(* CoDeSys 2.3 library: Smi_plc.lib *)

(* Global variable list: Error_Codes *)
VAR_GLOBAL CONSTANT
	(** @name Error Return Codes SMI
		Error code MOD 1000: are the error numbers below, see Smi_ExtractLibErr()
	@{ *)
	Smi_ERC_ConnId_InUse:	DINT := 2; (**< State connection-handle in use, communication cannot be reinitialized or closed *)
	Smi_ERC_Busy:			DINT := 1; (**< State busy, wait till finished *)
	Smi_ERC_Ok:				DINT := 0; (**< State OK, block can perform new order *)
	Smi_ERC_OtherError:		DINT := -1; (**< Other error not forward *)
	Smi_ERC_ParmInvalid:	DINT := -2; (**< Parameters are invalid *)
	Smi_ERC_NoCard:			DINT := -3; (**< Card not found / existing *)
	Smi_ERC_GetModNb:		DINT := -4; (**< Can't get Module-Number *)
	Smi_ERC_GetVal:			DINT := -5; (**< GetValue unsuccessfull *)
	Smi_ERC_SetVal:			DINT := -6; (**< SetValue unsuccessfull *)
	Smi_ERC_NoHandle:		DINT := -7; (**< Invalid Connection/Handle *)
	Smi_ERC_NoSelf:			DINT := -8; (**< User not identified as PLC project *)
	Smi_ERC_NoMemory:		DINT := -10; (**< No free Memory *)
	Smi_ERC_Internal:		DINT := -11; (**< Internal error on RPC-Requester *)
	Smi_ERC_RepQAdd:		DINT := -12; (**< Reply-Queue full *)
	Smi_ERC_Timeout:		DINT := -13; (**< Communication time exceeded/Communication timeout *)
	Smi_ERC_SendCall:		DINT := -14; (**< Can't send request *)
	Smi_ERC_GetBlk:			DINT := -15; (**< GetBlock unsuccessfull *)
	Smi_ERC_SetBlk:			DINT := -16; (**< SetBlock unsuccessfull *)
	Smi_ERC_GetFnLib:		DINT := -17; (**< Can't get Function-Library *)
	Smi_ERC_WrongVers:		DINT := -18; (**< Wrong Version of MSys *)
	Smi_ERC_ResultLen:		DINT := -19; (**< Reply-Size does not match *)
	Smi_ERC_GetValLst:		DINT := -20; (**< GetValLst unsuccessfull *)
	Smi_ERC_SetValLst:		DINT := -21; (**< SetValLst unsuccessfull *)
	Smi_ERC_GetAddr:		DINT := -22; (**< GetAddress unsuccessfull *)
	Smi_ERC_ModInfo:		DINT := -24; (**< ModInfo-Rpc unsuccessfull *)
	Smi_ERC_AppInfo:		DINT := -25; (**< AppInfo-Rpc unsuccessfull *)
	Smi_ERC_SemCreate:		DINT := -26; (**< Failed to create semaphore *)
	Smi_ERC_PingInternal:	DINT := -30; (**< Intenal Error execute Ping *)
	Smi_ERC_RequestAccess:  DINT := -31; (**< RequestAccess-Rpc unsuccessfull *)
	Smi_ERC_ReleaseAccess:  DINT := -32; (**< RequestAccess-Rpc unsuccessfull *)
	Smi_ERC_LoginFail:		DINT := -95; (**< Authentification fail Name/Passwd *)
	(** @} *)

	(** @name Error Return Codes SVI
		Error code / -1000: SVI error number of counterpart, see Smi_ExtractSmiErr()
	@{ *)
	SVI_ERC_OK: 			DINT := 16#0; (**< O.K. *)
	SVI_ERC_UNDEF: 			DINT := 16#124; (**< FUNCTION NOT supported *)
	SVI_ERC_ADDR: 			DINT := 16#130; (**< SVI address NOT valid *)
	SVI_ERC_WRITE: 			DINT := 16#141; (**< SVI value NOT writable *)
	SVI_ERC_READ: 			DINT := 16#140; (**< SVI value NOT readable *)
	SVI_ERC_FAILED: 		DINT := 16#100; (**< Unspecified error *)
	SVI_ERC_OLDADDR: 		DINT := 16#17E; (**< Address NOT valid anymore *)
	SVI_ERC_NOMOD: 			DINT := 16#129; (**< Module NOT found *)
	SVI_ERC_BADNAME: 		DINT := 16#137; (**< Invalid varibale name *)
	SVI_ERC_PARM: 			DINT := 16#110; (**< Parameter NOT valid *)
	SVI_ERC_VARINUSE: 		DINT := 16#1AC; (**< Varibale already in use *)
	SVI_ERC_MBTRANS: 		DINT := 16#1AD; (**< This needs MB support *)
	SVI_ERC_MBNOBUFF: 		DINT := 16#1AE; (**< No buffer found *)
	SVI_E_NOMEM:            DINT := 16#123; (**< Not enough memory *)
	SVI_E_BADUSERLVL:  		DINT := 16#1EA; (**< Weak user level (deprecated: replaced by SVI_E_ACCDENIED) *)
	SVI_E_BADRANGE:     	DINT := 16#17C; (**< SVI value out of bounds *)
	SVI_E_ACCDENIED:    	DINT := 16#1E9; (**< Access denied *)
	SVI_E_DSIZE:        	DINT := 16#1C2; (**< Data size not valid, exceeds max size *)
	SVI_E_REDULOCK:     	DINT := 16#1F0; (**< Write access allowed only on primary CPU *)
	SVI_E_BADTYPE:      	DINT := 16#16A; (**< Wrong data type *)
	SVI_E_DLEN:         	DINT := 16#1F3; (**< Data length invalid *)
	SVI_E_BADSESS:          DINT := 16#19C; (**< Session ID not valid *)
	SBI_E_TIMEOUT2:         DINT := 16#127; (**< No answer from SW-Module *)
	(** @} *)

	(** @name Error Return Codes Socket-FBs
		Error code MOD 1000: are the error numbers below, see Smi_ExtractLibErr() \n
		Error code / -1000: VxWorks error number of the C function, see errno.h, Smi_ExtractSmiErr()
	@{ *)
	Smi_ERC_SockCreate:		DINT := -1; (**< Creation of socket failed *)
	Smi_ERC_SockClose:		DINT := -2; (**< Close of socket failed *)
	Smi_ERC_SockRead:		DINT := -3; (**< Read of socket failed *)
	Smi_ERC_SockWrite:		DINT := -4; (**< Write of socket failed *)
	Smi_ERC_SockBind:		DINT := -5; (**< bind of socket failed *)
	Smi_ERC_SockListen:		DINT := -6; (**< listen at socket init failed *)
	Smi_ERC_SockAccept:		DINT := -7; (**< accept at socket init failed *)
	Smi_ERC_SockConnect:	DINT := -8; (**< Connect failed *)
	Smi_ERC_SockInvProt:	DINT := -9; (**< Invalid protocoll *)
	Smi_ERC_SockShutdown:	DINT := -10; (**< Shutdown failed *)
	Smi_ERC_SockSetOpt:		DINT := -11; (**< Set option of socket failed *)
	(** @} *)

	(** @name Error Return Codes Retain
		for Smi_RetainExport() or its SMI-Call
	@{ *)
	RETEXP_E_UNKNOWNERROR: 		DINT := 100; (**< Unexpected error. *)
	RETEXP_E_NOMEMORY: 			DINT := 102; (**< Not enough memory. *)
	RETEXP_E_MISSINGSTRUCTFILE: DINT := 103; (**< The retain structure couldn't be found. *)
	RETEXP_E_MISSINGDATAFILE: 	DINT := 104; (**< The retain data couldn't be found. *)
	RETEXP_E_RETAINDATACORRUPT: DINT := 105; (**< The retain data is corrupt. *)
	RETEXP_E_FILECREATIONFAILED:DINT := 106; (**< The export file couldn't be created/overwritten. *)
	(** @} *)
END_VAR

(* Global variable list: Global_Constants *)
(*
 PLC1131-Library with Functions for Communication by SVI and SMI
 Copyright: G.Bachmann GmbH, 1997-2011, Feldkirch - Austria
*)
VAR_GLOBAL CONSTANT
	(** @name Constants for 'VarCode'
	@{ *)
	Smi_MX_Code:			INT := 1; (**< MX marker *)
	Smi_MB_Code:			INT := 2; (**< MB marker *)
	Smi_MD_Code:			INT := 3; (**< MD marker *)
	Smi_MR_Code:			INT := 4; (**< MR marker *)
	Smi_MW_Code:			INT := 5; (**< MW marker *)
	Smi_RD_Code:			INT := 19; (**< RD marker *)
	Smi_GD_Code:			INT := 35; (**< GD marker *)
	(** @} *)

	(** @name Constants for 'ProtVers'
		in SMI_Connect(), SMI_Connect_NB(), SMI_Login(), SMI_Login_NB() and SMI_Ping() 
	@{ *)
	Smi_PROT_Tcp:			DWORD := 16#80000000; (**< Use TCP instead of UDP *)
	Smi_PROT_QSoap:			DWORD := 16#00004000; (**< Use bachmann proprietary SOAP as transport protocol (Quick SOAP)*)
	Smi_PROT_Ssl:           DWORD := 16#08000000; (**< Use SSL transport protocol *)
	Smi_PROT_PlainTxtPwd:   DWORD := 16#04000000; (**< Send plain text password *)
	(** @} *)

	(** @name Constants for 'TestLevel' and 'TestResult'
		in SMI_Ping(), SMI_PingEx()
	@{ *)
	Smi_LEVEL_IpPing:		WORD := 1; (**< IP-Ping *)
	Smi_LEVEL_AppInfo:		WORD := 2; (**< RES_APPINFO-Rpc *)
	Smi_LEVEL_ModInfo:		WORD := 4; (**< RES_MODINFO-Rpc *)
	Smi_LEVEL_RpcPing:		WORD := 8; (**< Rpc-Ping to Module *)
	Smi_LEVEL_FtpCheck:		WORD := 16; (**< Ftp-Test-Login *)
	(** @} *)

	(** @name Constants for 'AppState'
		in SMI_Ping(), SMI_PingEx()
	@{ *)
	Smi_RESSTAT_Run:		DWORD := 1; (**< Module is running *)
	Smi_RESSTAT_Error:		DWORD := 2; (**< Module is in error *)
	Smi_RESSTAT_Stop:		DWORD := 3; (**< Module stopped *)
	Smi_RESSTAT_Init:		DWORD := 4; (**< Module is in init *)
	Smi_RESSTAT_Deinit:		DWORD := 5; (**< Module is in deinit *)
	Smi_RESSTAT_Eoi:		DWORD := 6; (**< Module is waiting *)
	(** @} *)

	(** @name Available SMI Commands
		of SMI_Command()
	@{ *)
	CMD_SMI_PROC_NULL:			DWORD := 0; (**< SMI-Ping *)
	CMD_SMI_PROC_DEINIT:		DWORD := 4; (**< Uninstall module *)
	CMD_SMI_PROC_RESET:			DWORD := 6; (**< Reset module *)
	CMD_SMI_PROC_NEWCFG:		DWORD := 8; (**< New configuration of module *)
	CMD_SMI_PROC_ENDOFINIT:		DWORD := 14; (**< Signal end of init *)
	CMD_SMI_PROC_STOP:			DWORD := 18; (**< Stop module *)
	CMD_SMI_PROC_RUN:			DWORD := 20; (**< Start module *)
    CMD_PLC_PROC_RETAINEXPORT:  DWORD := 1546; (**< Export RETAIN data FOR an application *)
	(** @} *)

	(** @name Constants of Sockets
		of Smi_SOCK_ClientOpen(), Smi_SOCK_ClientOpen_NB(), Smi_SOCK_ServerOpen(), Smi_SOCK_ServerOpen_NB()
	@{ *)
	Smi_SOCK_ProtoTCP:		DWORD :=  6; (**< Protocol AF_INET/TCP *)
	Smi_SOCK_ProtoUDP:		DWORD := 17; (**< Protocol AF_INET/UDP *)
	Smi_SOCK_ModeDirect:	DINT := 0; (**< Parameter for mode: direct operation *)
	Smi_SOCK_ModeNoWait:	DINT := 2; (**< Parameter for mode: Smi_SOCK_Read() returns immediatly *)
	Smi_SOCK_SO_KEEPALIVE:	DINT := 16#0008; (**< keep connections alive, 1(on=default)/0(off) *)
 	Smi_SOCK_SO_BROADCAST:	DINT := 16#0020; (**< permit sending to multiple destination 1(on)/0(off) *)
 	Smi_SOCK_SO_SNDBUFF:	DINT :=	16#1001; (**< specifying the size of the send buffer *)
 	Smi_SOCK_SO_RCVBUFF:	DINT := 16#1002; (**< specifying the size of the beceive buffer *)
	(** @} *)
END_VAR

(* Global variable list: Library_Info *)
VAR_GLOBAL CONSTANT
	SMI_PLC_LIBVER					:	STRING(16) 	:=	'V1.36 Release';	(* Version String *)
    SMI_PLC_MMPREADY                :   BOOL        :=  TRUE;               (* MMP Ready *)
END_VAR

(* Data type *)
(*
	structure to specify 64 Bit Smi Address Handle
*)
TYPE SMI_ADDR
STRUCT
	Addr1:		DWORD;		(* SmiAddr Handle 1st 32 Bit *)
	Addr2:		DWORD;		(* SmiAddr Handle 2nd 32 Bit *)
END_STRUCT
END_TYPE

(* Data type *)
(*
	return-structure of Smi_GetConnStatus
*)
TYPE SMI_RETCONNSTAT
STRUCT
	RetCode:	DINT;		(* Success (0) - or Error-Code (<0) *)
	CpuNb:		DINT;		(* CPU-Number *)
	ModuleNb:	DWORD;		(* Module-Number (SMI-Master) *)
	PLibAddr:	DWORD;		(* SVI-Function-Lib-Pointer *)
	UseCount:	DINT;		(* Number of pending requests (FBs) *)
	ErrorCode:	DINT;		(* Last Error on Connection *)
	FnGetStat:	DINT;		(* Read/Write-Get-Status *)
	FnRdyStat:	DINT;		(* Read/Write-Ready-Status *)
END_STRUCT
END_TYPE

(* Data type *)
(* This structure is filled at Smi_SOCK_ClientOpen and
   Smi_SOCK_ServerOpen *)
TYPE SMI_SOCK_CONTROL :
STRUCT
	ProtType:		DWORD;
	Port:			WORD;
	IpAddr:			DINT;
	Socket:			DWORD;
    ServerSocket:   DWORD;
END_STRUCT
END_TYPE

(* Data type *)
(*
	structure to specify a Marker-Variable
*)
TYPE VAR_ADDR
STRUCT
	VarCode:	DWORD;		(* Marker-Type 1:MX, 2:MB, 3:MD, 4:MR, 5:MW *)
	VarIndex:	DWORD;		(* Index of Marker *)
END_STRUCT
END_TYPE

(* POU GetREALasDWORD, IL *)
(**
@brief Return a REAL from contents of DWORD
@param[in] dw Input variable
@return REAL interpreted value
*)
FUNCTION GetREALasDWORD : REAL
VAR_INPUT
	dw: DWORD;
END_VAR
	LD		0
END_FUNCTION

(* POU SetREALasDWORD, IL *)
(**
@brief Returns REAL 'x' casted to a DWORD
@param[in] x REAL value
@return DWORD-coded value
*)
FUNCTION SetREALasDWORD : DWORD
VAR_INPUT
	x: REAL;
END_VAR
LD 0
END_FUNCTION

(* POU Smi_BuildNbFromIP, IL *)
(**
@brief Makes a CPU-Number representing an IP-Address
@param[in] b1 1. Byte of the IP adress
@param[in] b2 2. Byte of the IP adress
@param[in] b3 3. Byte of the IP adress
@param[in] b4 4. Byte of the IP adress
@return Coded IP address (CPU number)
*)
FUNCTION Smi_BuildNbFromIP : DINT
VAR_INPUT
	b1: BYTE;
	b2: BYTE;
	b3: BYTE;
	b4: BYTE;
END_VAR
LD 0
END_FUNCTION

(* POU Smi_BuildNbFromName, IL *)
(**
@brief Makes a CPU-Number for a Host-Name or an IP-String
@param[in] Name IP-Adresse in octet-Notation (e.g. 192.9.200.30)
@return Coded IP address (CPU number). The value is to be transferred 
	to the input parameter CpuNb of the function blocks SMI_Connect() and SMI_CheckIp_NB appropriate. 
*)
FUNCTION Smi_BuildNbFromName : DINT
VAR_INPUT
	Name : STRING(23);
END_VAR
	LD		0
END_FUNCTION

(* POU SMI_BuildNbFromName_NB, ST *)
(**
@brief Makes a CPU-Number for a Host-Name or an IP-String, non-blocking.
@param[in] Req If false only state is returned. If true and state is not busy,
    a command is done.
@param[in] Name IP-Address in Octet-Notation  '192.9.100.10' or 'hostname'
@param[out] Done TRUE if ready
@param[out] Error TRUE in case of error
@param[out] Status Error code in case of error 
    - <tt>#Smi_ERC_Ok</tt>OK. <tt>Done = TRUE</tt>, <tt>ConnId</tt> valid
    - <tt>#Smi_ERC_Busy</tt>Completion/response is pending, <tt>CpuNb </tt> is not available
    - <tt>#Smi_ERC_OtherError</tt>Name or IP address is invalid, CpuNb is not available.
@param[out] CpuNb Coded IP address (CPU number). The value is to be transferred to the input 
	parameter CpuNb of the function blocks SMI_Connect(), SMI_Connect_NB(), SMI_Login(), SMI_Login_NB() 
	and SMI_CheckIp_NB appropriate.
*)
FUNCTION_BLOCK SMI_BuildNbFromName_NB
VAR_INPUT
	Req:			BOOL;
    Name:       	STRING(63);
END_VAR
VAR_OUTPUT
	Done: 		BOOL;
	Error: 		BOOL;
	Status: 	DINT;
	CpuNb: 		DINT;
END_VAR
VAR
	Pltd: DWORD;
END_VAR
;
END_FUNCTION_BLOCK

(* POU SMI_Call, IL *)
(**
@brief This function block is used to send SMI-messages. Timeout is
    interal set to 2000ms and no retries.
  Note: The size of the in and out buffer are limited to SMI_DATALEN.
@param[in] Req If false only state is returned. If true and state is not busy,
    a command is done.
@param[in] ConnId Connection identifier for the connection. 
           The connection identifier can be determined with SMI_Login() or SMI_Connect().
@param[in] SmiFcnNumber Specifies which SMI functions should be executed. 
    General SMI functions can be called
@param[in] DataSend Address of send buffer, use ADR(). Specification of the transmit 
    buffer Maximum size: 1996 bytes.
@param[in] DataSendLen Length of send buffer. 
    Specification of the transmit buffer Maximum size: 1996 bytes. 
@param[in] DataRec Address of receive buffer, use ADR(). 
    Specification of the receive buffer Maximum size: 1996 bytes. 
@param[in] DataRecLen Specification of the receive buffer Maximum size: 1996 bytes.
@param[out] State Error code in case of error 
    - <tt>#Smi_ERC_Ok</tt> OK
    - <tt>#Smi_ERC_Busy</tt> Completion/response is pending
    - <tt>Smi_ERC_*</tt> Error codes are negative
@param[out] RecLen Specification of the number of bytes received
    The minimum of <tt>DataRecLen</tt> and RecLen is copied to the receive buffer.
*)
FUNCTION_BLOCK SMI_Call
VAR_INPUT
	Req:			BOOL;
	ConnId:			DWORD;
	SmiFcnNumber:	DWORD;
	DataSend:		DWORD;
	DataSendLen:	DINT;
	DataRec:		DWORD;
	DataRecLen:		DINT;
END_VAR
VAR_OUTPUT
	State: 			DINT;
	RecLen:			DINT;
END_VAR
VAR
	fi: 			UDINT;
END_VAR
	LD		0
END_FUNCTION_BLOCK

(* POU SMI_CheckIp_NB, ST *)
(**
@brief non-blocking FB to check if an IP is occupied. (on MPC only)
@param[in] Req Request enable
@param[in] EthCard To use Ethernet interface (starting with 0).
@param[in] CpuNb Coded IP address (CPU number).\n
    The IP address must be coded beforehand. (Smi_BuildNbFromIP or Smi_BuildNbFromName). 
@param[in] Timeout The parameter is used to indicate the response latency. By Timeout = 0 
	is wait for 3 seconds. [ms]
@param[out] Mac Contains the MAC address of the desired host when parameter Done is set.
@param[out] MacHexStr Contains the MAC address in string format when parameter Done is set.
@param[out] Done TRUE if ready
@param[out] Error TRUE in case of error
@param[out] Status Error code in case of error 
    - <tt>#Smi_ERC_Ok</tt> OK. <tt>Done = TRUE</tt>, <tt>Mac</tt> valid
    - <tt>#Smi_ERC_Busy</tt> Completion/response is pending, <tt>Mac</tt> is not available
    - <tt>Smi_ERC_*</tt> Error codes are negative. <tt>Error = TRUE;</tt> Mac not available. 
*)
FUNCTION_BLOCK SMI_CheckIp_NB
VAR_INPUT
	Req: BOOL;
	EthCard: DINT;
	CpuNb: DINT;
	Timeout: TIME;
END_VAR
VAR_OUTPUT
	Mac: ARRAY[1..6] OF BYTE;
	MacHexStr: STRING(17);
	Done: BOOL;
	Error: BOOL;
	Status: DINT;
END_VAR
VAR
	hJob: DWORD;
END_VAR
;
END_FUNCTION_BLOCK

(* POU SMI_CloseConnect, ST *)
(**
@brief close a connection to a remote host opened with SMI_Connect or SMI_Login
@param[in] Req Request enable
@param[in] ConnId Transfer of the connection identifier for the connection.
    The identifier can be determined with SMI_Login() or SMI_Connect().
@param[out] Done TRUE if ready
@param[out] Error TRUE in case of error
@param[out] Status Error code in case of error
    - <tt>#Smi_ERC_Ok</tt> OK. <tt>Done = TRUE</tt>
    - <tt>Smi_ERC_*</tt> Error codes are negative
*)
FUNCTION_BLOCK SMI_CloseConnect
VAR_INPUT
	Req: BOOL;
	ConnId: DWORD;
END_VAR
VAR_OUTPUT
	Done: BOOL;
	Error: BOOL;
	Status: DINT;
END_VAR
VAR
END_VAR
;
END_FUNCTION_BLOCK

(* POU SMI_Command, IL *)
(**
@brief This function block is used to send SMI-messages. Timeout is
    interal set to 2000ms and no retries.
@param[in] Req request-enable: if false only state is returned
@param[in] ConnId Connection identifier for the connection. 
           The connection identifier can be determined with SMI_Login() or SMI_Connect().
@param[in] SmiFcnNumber SMI function to be executed. Allowed functions
    - <tt>#CMD_SMI_PROC_NULL</tt>
    - <tt>#CMD_SMI_PROC_DEINIT</tt>
    - <tt>#CMD_SMI_PROC_RESET</tt>
    - <tt>#CMD_SMI_PROC_NEWCFG</tt>
    - <tt>#CMD_SMI_PROC_ENDOFINIT</tt>
    - <tt>#CMD_SMI_PROC_STOP</tt>
    - <tt>#CMD_SMI_PROC_RUN</tt>
@param[in] ModuleName Name of target module, has to be the same as in SMI_Connect or
    SMI_Login
@param[out] Error If TRUE error occured
@param[out] State Error code in case of error 
    - <tt>#Smi_ERC_Ok</tt> OK
    - <tt>#Smi_ERC_Busy</tt> Completion/response is pending
    - <tt>Smi_ERC_*</tt> Error codes are negative
*)
FUNCTION_BLOCK SMI_Command
VAR_INPUT
	Req			: BOOL;
	ConnId		: DWORD;
	SmiFcnNumber :	DWORD;
	ModuleName 	: STRING(11);
END_VAR
VAR_OUTPUT
	Error	 	: BOOL;
	State	 	: DINT;
END_VAR
VAR
	fi: UDINT;
END_VAR
	LD		0
END_FUNCTION_BLOCK

(* POU SMI_Connect, IL *)
(**
@brief Build/init Connection to named SMI-Module on local or remote CPU
@param[in] CpuNb With the parameter the IP address of the CPU of the communication partner will be transferred. 
@param[in] MasterName With the parameter, the name of the partner module (communication partner) will be transferred.
@param[in] Reinit The parameter must be set if a previously-established connection should be renewed
@param[in] ProtVers The parameter is used to specify the RPC protocol version to be used. This input must be used 
	when SMI is used for the connection.
    The possible RPC protocol versions depend on the communication partner (process value supplier). This input can 
	be used to switch the protocol to TCP using the entry SMI_PROT_Tcp (OR link with the protocol version). The UDP 
	protocol is used without OR link with PROT_Tcp. System modules/handler and PLC projects based on M1 software 
	V1.00 release and the simultaneously-created available controller modules generally use RPC protocol version 2. 
	Consequently, the value 2 has to be indicated at the parameter ProtVers.
@param[out] Done TRUE if ready
@param[out] Error TRUE in case of error
@param[out] Status Error code in case of error
    - <tt>#Smi_ERC_Ok</tt> OK. <tt>Done = TRUE</tt>, <tt>ConnId</tt> valid
    - <tt>#Smi_ERC_Busy</tt> Completion/response is pending, <tt>ConnId</tt> is not available
    - <tt>#Smi_ERC_ConnId_InUse</tt> Reinitialization presently not possible; communication in process
    - <tt>Smi_ERC_*</tt> Error codes are negative. 
@param[out] ConnId Connection-Identifier
*)
FUNCTION_BLOCK SMI_Connect
VAR_INPUT
	CpuNb: 		DINT;
	MasterName: STRING(15);
	Reinit: 	BOOL;
	ProtVers: 	DWORD;
END_VAR
VAR_OUTPUT
	Done: 		BOOL;
	Error: 		BOOL;
	Status: 	DINT;
	ConnId: 	DWORD;
END_VAR
VAR
	fi: UDINT;
END_VAR
LD 0
END_FUNCTION_BLOCK

(* POU SMI_Connect_NB, IL *)
(**
@brief Non blocking version of SMI_Connect, Build/init Connection to named SMI-Module on local or remote CPU
@param[in] CpuNb With the parameter the IP address of the CPU of the communication partner will be transferred.
    see Smi_BuildNbFromName()
@param[in] MasterName With the parameter, the name of the partner module (communication partner) will be transferred.
@param[in] Reinit The parameter must be set if a previously-established connection should be renewed
@param[in] ProtVers The parameter is used to specify the RPC protocol version to be used. This input 
	must be used when SMI is used for the connection.\n
    The possible RPC protocol versions depend on the communication partner (process value supplier). This input can 
	be used to switch the protocol to TCP using the entry SMI_PROT_Tcp (OR link with the protocol version). The UDP 
	protocol is used without OR link with PROT_Tcp. System modules/handler and PLC projects based on M1 software 
	V1.00 release and the simultaneously-created available controller modules generally use RPC protocol version 2. 
	Consequently, the value 2 has to be indicated at the parameter ProtVers.
@param[out] Done TRUE if ready
@param[out] Error TRUE in case of error
@param[out] Status Error code in case of error
    - <tt>#Smi_ERC_Ok</tt> OK. <tt>Done = TRUE</tt>, <tt>ConnId</tt> valid
    - <tt>#Smi_ERC_Busy</tt> Completion/response is pending, <tt>ConnId</tt> is not available
    - <tt>#Smi_ERC_ConnId_InUse</tt> Reinitialization presently not possible; communication in process
    - <tt>Smi_ERC_*</tt> Error codes are negative. 
@param[out] ConnId Connection-Identifier
*)
FUNCTION_BLOCK SMI_Connect_NB
VAR_INPUT
	CpuNb: 		DINT;
	MasterName: STRING(15);
	Reinit: 	BOOL;
	ProtVers: 	DWORD;
END_VAR
VAR_OUTPUT
	Done: 		BOOL;
	Error: 		BOOL;
	Status: 	DINT;
	ConnId: 	DWORD;
END_VAR
VAR
	fi: UDINT;
	Pltd: DWORD;
	uState: DWORD;
END_VAR
LD 0
END_FUNCTION_BLOCK

(* POU Smi_ExtractLibErr, ST *)
(**
@brief The functions and functionblocks of the SMI-library return
    a 'packed' error-code/status which encodes two specific errors.

    This function extracts the library-error of the encoded error.
    The library-error is generated in the SMI-library directly,
    eg through checking the input-parameters.

    The library-error can be compared against the Smi_ERC_xxx-constants.

@param[in] Error Error returned by the Smi_-function or -functionblock
@return DINT, see description
*)
FUNCTION Smi_ExtractLibErr : DINT
VAR_INPUT
	Error: DINT;
END_VAR
VAR
END_VAR
;
END_FUNCTION

(* POU Smi_ExtractSmiErr, ST *)
(**
@brief Functions and functions of the SMI-library, return
    a 'packed' error-code/status which encodes two specific errors.

    This function extracts the SMI-error (error/return-value
    of the SMI-reply-message) of the encoded error.
@param[in] Error error returned by the Smi_-function or -functionblock
@return DINT, see description
*)
FUNCTION Smi_ExtractSmiErr : DINT
VAR_INPUT
	Error: DINT;
END_VAR
VAR
END_VAR
;
END_FUNCTION

(* POU SMI_GetAddr, ST *)
(**
@brief Gets the SMI-Address-Handle of the Symbolic SVI-Object from
    SMI-Module
@param[in] Req Request enable
@param[in] ConnId Transfer of the connection identifier for the connection. 
    The identifier can be determined with SMI_Login() or SMI_Connect(). 
@param[in] ValueName With the parameter the symbolic marker or process value 
    name is specified, for which the numeric address should be determined.
@param[out] Ndr TRUE if operation successfully completed/new data received
@param[out] Error TRUE in case of error
@param[out] Status see Smi_ERC_*
    - #Smi_ERC_Ok OK/Done
    - #Smi_ERC_Busy Completion/response is pending, result is not available
    - Smi_ERC_* Error occured
@param[out] Error TRUE in case of error
@param[out] SmiHandle Smi-Address-Handle of the Symbolic Object
*)
FUNCTION_BLOCK SMI_GetAddr
VAR_INPUT
	Req 		: BOOL;
	ConnId 		: DWORD;
	ValueName 	: STRING(63);
END_VAR
VAR_OUTPUT
	Ndr 		: BOOL;
	Error 		: BOOL;
	Status 		: DINT;
	SmiHandle	: SMI_ADDR;
END_VAR
VAR
	fi			: UDINT;
END_VAR
;
END_FUNCTION_BLOCK

(* POU SMI_GetAddress, ST *)
(**
@brief Gets Address of a Marker or Process-Value from SMI-Module
@param[in] Req Request enable
@param[in] ConnId Transfer of the connection identifier for the connection.
    The identifier can be determined with SMI_Login() or SMI_Connect().
@param[in] ValueName With the parameter the symbolic marker or process value name is specified, for which 
	the numeric address should be determined.
@param[out] Ndr TRUE if new data received
@param[out] Error TRUE in case of error
@param[out] Status Error code in case of error
    - <tt>#Smi_ERC_Ok</tt> OK. <tt>Ndr = TRUE</tt>, <tt>VAddr</tt> valid
    - <tt>#Smi_ERC_Busy</tt> Completion/response is pending, <tt>VAddr</tt> is not available
    - <tt>#Smi_ERC_ConnId_InUse</tt> Reinitialization presently not possible; communication in process
    - <tt>Smi_ERC_*</tt> Error codes are negative
@param[out] VAddr Marker- or Process-Value-Address
*)
FUNCTION_BLOCK SMI_GetAddress
VAR_INPUT
	Req : BOOL;
	ConnId : DWORD;
	ValueName : STRING(63);
END_VAR
VAR_OUTPUT
	Ndr : BOOL;
	Error : BOOL;
	Status : DINT;
	VAddr : VAR_ADDR;
END_VAR
VAR
	fi: UDINT;
END_VAR
;
END_FUNCTION_BLOCK

(* POU SMI_GetBlk, ST *)
(**
@brief Reads a String or Stream of Bytes from SMI-Module
@param[in] Req Request enable
@param[in] ConnId Transfer of the connection identifier for the connection.
    The identifier to be transferred can be determined with SMI_Login() or SMI_Connect().
@param[in] SmiHandle The start address of the marker block to be read or the SVI variable.
    This is determined by SMI_GetAddr().
@param[in] Addr Address of a data range into which the values are read.
@param[in] Length Length of the data range. If a block of markers is read, the value byte 
	stream is 4 byte aligned. 
@param[out] Ndr TRUE if operation successfully completed/new data received
@param[out] Error TRUE in case of error
@param[out] Status see Smi_ERC_*
    - #Smi_ERC_Ok OK/Done
    - #Smi_ERC_Busy Completion/response is pending, result is not available
    - Smi_ERC_* Error occured
@param[out] NRead number of bytes read
*)
FUNCTION_BLOCK SMI_GetBlk
VAR_INPUT
	Req			: BOOL;
	ConnId		: DWORD;
	SmiHandle	: SMI_ADDR;
	Addr 		: DWORD;
	Length		: UINT;
END_VAR
VAR_OUTPUT
	Ndr			: BOOL;
	Error	 	: BOOL;
	Status		: DINT;
	NRead		: UINT;
END_VAR
VAR
	fi			: UDINT;
END_VAR
;
END_FUNCTION_BLOCK

(* POU Smi_GetConnStatus, IL *)
(**
@brief Gets information on Status of Connection
@param[in] ConnId Transfer of the connection identifier for the connection. The identifier can be determined 
	with SMI_Login() or SMI_Connect(). 
@retval SMI_RETCONNSTAT.RetCode = #Smi_ERC_Ok: Everything OK.
@retval SMI_RETCONNSTAT.RetCode = #Smi_ERC_NoSelf: User not identified as PLC project.
*)
FUNCTION Smi_GetConnStatus : SMI_RETCONNSTAT
VAR_INPUT
	ConnId: DWORD;
END_VAR
LD 0
END_FUNCTION

(* POU Smi_GetOwnIPAddr, IL *)
(**
@brief Makes a Number representing the own IP-Address
@param[in] EthCard ethernet-interface (0 or 1)
@return Coded IP address (CPU number)
*)
FUNCTION Smi_GetOwnIPAddr : DINT
VAR_INPUT
	EthCard:	DINT;
END_VAR
LD 0
END_FUNCTION

(* POU SMI_GetVal, ST *)
(**
@brief Reads a single SVI-Var-Object from a SMI-Module
@param[in] Req Request enable
@param[in] ConnId Transfer of the connection identifier for the connection.
    The identifier to be transferred can be determined with SMI_Login() or SMI_Connect().
@param[in] SmiHandle 64-Bit Smi Object Handle/process value's address
    This is determined by SMI_GetAddr().
@param[out] Ndr TRUE if operation successfully completed/new data received
@param[out] Error TRUE in case of error
@param[out] Status see Smi_ERC_*
    - #Smi_ERC_Ok OK/Done
    - #Smi_ERC_Busy Completion/response is pending, result is not available
    - Smi_ERC_* Error occured
@param[out] Value Read-Value 32-Bit Format
*)
FUNCTION_BLOCK SMI_GetVal
VAR_INPUT
	Req			: BOOL;
	ConnId		: DWORD;
	SmiHandle	: SMI_ADDR;
END_VAR
VAR_OUTPUT
	Ndr			: BOOL;
	Error		: BOOL;
	Status		: DINT;
	Value		: DWORD;
END_VAR
VAR
	fi			: UDINT;
END_VAR
;
END_FUNCTION_BLOCK

(* POU Smi_GetValFn, IL *)
(**
@brief Reads Smi Objekt (specified by Smi Address) from SMI-Module.
    Implementation: an Rpc-Request is done, read may be BUSY
    until Rpc-Reply is received.
@param[in] ConnId Transfer of the connection identifier for the connection.
    The identifier to be transferred can be determined with SMI_Login() or SMI_Connect().
@param[in] SmiAddr Address of 64-Bit Smi Object Handle/process value's address
@param[in] ValAddr Address to store read Value
@retval #Smi_ERC_Ok OK
@retval #Smi_ERC_Busy Completion/response is pending; read value not available yet
@retval #Smi_ERC_ConnId_InUse Other function is being processed; communication in process
@retval Smi_ERC_* Error codes are negative 
*)
FUNCTION Smi_GetValFn : DINT
VAR_INPUT
	ConnId		: DWORD;
	SmiAddr		: DWORD;
	ValAddr		: DWORD;
END_VAR
LD 0
END_FUNCTION

(* POU SMI_GetValLst, IL *)
(**
@brief Reads a List of Smi-Objects from SMI-Module
@param[in] Req Request enable
@param[in] ConnId Transfer of the connection identifier for the connection.
    The identifier to be transferred can be determined with SMI_Login() or SMI_Connect().
@param[in] SmiHandleF List of Smi-Address-Handles. This is determined by SMI_GetAddr(). 
@param[in] NumberOf Number of addresses, maximal 64
@param[out] Ndr TRUE if operation successfully completed/new data received
@param[out] Error TRUE in case of error
@param[out] Status see Smi_ERC_*
    - #Smi_ERC_Ok OK/Done
    - #Smi_ERC_Busy Completion/response is pending, result is not available
    - Smi_ERC_* Error occured
@param[out] Rdf Data receive field
*)
FUNCTION_BLOCK SMI_GetValLst
VAR_INPUT
	Req			: BOOL;
	ConnId		: DWORD;
	SmiHandleF  : ARRAY[0..63] OF SMI_ADDR;
	NumberOf 	: DINT;
END_VAR
VAR_OUTPUT
	Ndr			: BOOL;
	Error	 	: BOOL;
	Status	 	: DINT;
	Rdf 		: ARRAY[0..63] OF DWORD;
END_VAR
VAR
	fi: UDINT;
END_VAR
LD 0
END_FUNCTION_BLOCK

(* POU Smi_GetVersion, ST *)
(**
@brief Returns the version string of the library. In simulation always
    '' is returned.
@param[in] dummy Unused parameter. 
@return Version string of the PLC library, e.g. V 1.03.01 Alpha, V 1.06.04 Beta, V1.04 Release.
*)
FUNCTION Smi_GetVersion : STRING(15)
VAR_INPUT
	dummy:		BOOL;
END_VAR
VAR
END_VAR
Smi_GetVersion := '';
END_FUNCTION

(* POU SMI_Login, IL *)
(**
@brief Build/init Connection to named SMI-Module with login on local 
    or remote CPU.
@param[in] CpuNb With the parameter the IP address of the CPU of the communication partner will be transferred. \n
    see: Smi_BuildNbFromName()
@param[in] MasterName With the parameter, the name of the partner module (communication partner) will be transferred.
@param[in] Reinit The parameter must be set if a previously-established connection should be renewed
@param[in] ProtVers The parameter is used to specify the RPC protocol version to be used. 
    This input must be used when SMI is used for the connection.\n
    The possible RPC protocol versions depend on the communication partner (process value supplier). This input can 
	be used to switch the protocol to TCP using the entry SMI_PROT_Tcp (OR link with the protocol version). The UDP 
	protocol is used without OR link with PROT_Tcp. System modules/handler and PLC projects based on M1 software 
	V1.00 release and the simultaneously-created available controller modules generally use RPC protocol version 2. 
	Consequently, the value 2 has to be indicated at the parameter ProtVers.
@param[in] LoginName With the parameter the login name is transferred.
@param[in] Password With the parameter the password that belongs to the login name is transferred.
    In case of an unencrypted password (Smi_PROT_PlainTxtPwd) the maximal password len is 16 (counterpart is older 
    than MSys 3.70 R) or 32 (counterpart is above MSys 3.70 R). In Case of an encrypted password the maximal len is 39. 
@param[out] Done TRUE if ready
@param[out] Error TRUE in case of error
@param[out] Status Error code in case of error
    - <tt>#Smi_ERC_Ok</tt> OK. <tt>Done = TRUE</tt>, <tt>ConnId</tt> valid
    - <tt>#Smi_ERC_Busy</tt> Completion/response is pending, <tt>ConnId</tt> is not available
    - <tt>#Smi_ERC_ConnId_InUse</tt> Reinitialization presently not possible; communication in process
    - <tt>Smi_ERC_*</tt> Error codes are negative. 
@param[out] ConnId Connection-Identifier
*)
FUNCTION_BLOCK SMI_Login
VAR_INPUT
	CpuNb: 		DINT;
	MasterName: STRING(15);
	Reinit: 	BOOL;
	ProtVers: 	DWORD;
	LoginName:	STRING(19);
	Password:	STRING(39);
END_VAR
VAR_OUTPUT
	Done: 		BOOL;
	Error: 		BOOL;
	Status: 	DINT;
	ConnId: 	DWORD;
END_VAR
VAR
	fi: UDINT;
END_VAR
	LD		0
END_FUNCTION_BLOCK

(* POU SMI_Login_NB, IL *)
(**
@brief Non-blocking version of SMI_Login. 
    Build/init Connection to named SMI-Module with login on local or remote CPU.
@param[in] CpuNb With the parameter the IP address of the CPU of the communication partner will be transferred. \n
    see: Smi_BuildNbFromName()
@param[in] MasterName With the parameter, the name of the partner module (communication partner) will be transferred.
@param[in] Reinit The parameter must be set if a previously-established connection should be renewed
@param[in] ProtVers The parameter is used to specify the RPC protocol version to be used. 
    This input must be used when SMI is used for the connection.\n
    The possible RPC protocol versions depend on the communication partner (process value supplier). This input can 
	be used to switch the protocol to TCP using the entry SMI_PROT_Tcp (OR link with the protocol version). The UDP 
	protocol is used without OR link with PROT_Tcp. System modules/handler and PLC projects based on M1 software V1.00 
	release and the simultaneously-created available controller modules generally use RPC protocol version 2. Consequently, 
	the value 2 has to be indicated at the parameter ProtVers.
@param[in] LoginName With the parameter the login name is transferred.
@param[in] Password With the parameter the password that belongs to the login name is transferred.
    In case of an unencrypted password (Smi_PROT_PlainTxtPwd) the maximal password len is 16 (counterpart is older 
    than MSys 3.70 R) or 32 (counterpart is above MSys 3.70 R). In Case of an encrypted password the maximal len is 39. 
@param[out] Done TRUE if ready
@param[out] Error TRUE in case of error
@param[out] Status Error code in case of error
    - <tt>#Smi_ERC_Ok</tt> OK. <tt>Done = TRUE</tt>, <tt>ConnId</tt> valid
    - <tt>#Smi_ERC_Busy</tt> Completion/response is pending, <tt>ConnId</tt> is not available
    - <tt>#Smi_ERC_ConnId_InUse</tt> Reinitialization presently not possible; communication in process
    - <tt>Smi_ERC_*</tt> Error codes are negative. 
@param[out] ConnId Connection-Identifier
*)
FUNCTION_BLOCK SMI_Login_NB
VAR_INPUT
	CpuNb: 		DINT;
	MasterName: STRING(15);
	Reinit: 	BOOL;
	ProtVers: 	DWORD;
	LoginName:	STRING(19);
	Password:	STRING(39);
END_VAR
VAR_OUTPUT
	Done: 		BOOL;
	Error: 		BOOL;
	Status: 	DINT;
	ConnId: 	DWORD;
END_VAR
VAR
	fi: UDINT;
	Pltd : DWORD;
	uState: DWORD;
END_VAR
	LD		0
END_FUNCTION_BLOCK

(* POU SMI_Ping, IL *)
(**
@brief Test Communication to CPU/Host or named SMI-Module on local
    or remote CPU.
@param[in] Req Request enable
@param[in] CpuNb With the parameter the IP address of the CPU of the communication partner will be transferred.\n
    see Smi_BuildNbFromName()
@param[in] ModuleName With the parameter the IP address of the CPU of the communication partner is transferred. 
    Relevance depends on <tt>TestLevel</tt>.
@param[in] ProtVers The parameter <tt>ProtVers</tt> is used to specify the RPC protocol version used (usually 2).
@param[in] TestLevel Use this parameter to specify what should be tested, or the scope in which the test should be executed. 
    For this the constants Smi_LEVEL_* are available. These can also be combined.
@param[out] Done TRUE if ready
@param[out] Error TRUE in case of error
@param[out] Status Error code in case of error 
    - <tt>#Smi_ERC_Ok</tt> OK. <tt>Done = TRUE</tt>, Result valid
    - <tt>#Smi_ERC_Busy</tt> Completion/response is pending, Result is not available
    - <tt>#Smi_ERC_GetModNb</tt> The RES_MODNB-Rpc was not successful.
    - <tt>#Smi_ERC_Timeout</tt> The communication partner (the CPU, the HOST, the software module) does not respond or 
        cannot be accessed.
    - <tt>#Smi_ERC_WrongVers</tt> SMI_Ping() does not function with this version of MSys; SMI_Ping() cannot be used until 
        MSys = V1.02 is used.
    - <tt>#Smi_ERC_ResultLen</tt> The returned data is inadequate or incompletely received.
    - <tt>#Smi_ERC_ModInfo</tt> The RES_MODINFO-Rpc was not successful.
    - <tt>#Smi_ERC_AppInfo</tt> The RES_APPINFO-Rpc was not successful.
@param[out] TestResult Degree of successfull Test: <tt>Smi_LEVEL_*</tt>
@param[out] AppState State of Module or Application <tt>Smi_RESSTAT_*</tt>
*)
FUNCTION_BLOCK SMI_Ping
VAR_INPUT
	Req: BOOL;
	CpuNb: DINT;
	ModuleName: STRING(15);
	ProtVers: DWORD;
	TestLevel: WORD;
END_VAR
VAR_OUTPUT
	Done: BOOL;
	Error: BOOL;
	Status: DINT;
	TestResult: WORD;
	AppState: DWORD;
END_VAR
VAR
	Pltd: DWORD;
END_VAR
LD 0
END_FUNCTION_BLOCK

(* POU SMI_PingEx, IL *)
(**
@brief Test Communication to CPU/Host or named SMI-Module on local or remote CPU. 
    Can handle the Connection-ID from SMI_Connect() or SMI_Login().
@param[in] Req Request enable
@param[in] ConnId With the parameter the connection ID that was received from the function 
    SMI_Connect() or SMI_Login(), is transferred. 
@param[in] TestLevel Use this parameter to specify what should be tested, or the scope in 
    which the test should be executed. For this the constants <tt>SMI_LEVEL...</tt> are available. 
    These can also be combined.
@param[out] Done TRUE if ready
@param[out] Error TRUE in case of error
@param[out] Status Error code in case of error 
    - <tt>#Smi_ERC_Ok</tt> OK. <tt>Done = TRUE</tt>, Result valid
    - <tt>#Smi_ERC_Busy</tt> Completion/response is pending, Result is not available
    - <tt>#Smi_ERC_GetModNb</tt> The RES_MODNB-Rpc was not successful.
    - <tt>#Smi_ERC_Timeout</tt> The communication partner (the CPU, the HOST, the software module) does not respond or 
        cannot be accessed.
    - <tt>#Smi_ERC_WrongVers</tt> SMI_Ping() does not function with this version of MSys; SMI_Ping() cannot be used until 
        MSys = V1.02 is used.
    - <tt>#Smi_ERC_ResultLen</tt> The returned data is inadequate or incompletely received.
    - <tt>#Smi_ERC_ModInfo</tt> The RES_MODINFO-Rpc was not successful.
    - <tt>#Smi_ERC_AppInfo</tt> The RES_APPINFO-Rpc was not successful.
@param[out] TestResult Degree of successfull Test: <tt>Smi_LEVEL_*</tt>
@param[out] AppState State of Module or Application <tt>Smi_RESSTAT_*</tt>
*)
FUNCTION_BLOCK SMI_PingEx
VAR_INPUT
	Req: BOOL;
	ConnId : DWORD;
	TestLevel: WORD;
END_VAR
VAR_OUTPUT
	Done: BOOL;
	Error: BOOL;
	Status: DINT;
	TestResult: WORD;
	AppState: DWORD;
END_VAR
VAR
	Pltd: DWORD;
END_VAR
LD 0
END_FUNCTION_BLOCK

(* POU Smi_Read, IL *)
(**
@brief Reads one marker (specified by VarCode/VarIndex) from a SMI-Module 
@param[in] ValAddr  Using the ADR operator, must be created from the variable 
                    that should contain the read value. This variable must comply with the 
                    specified market type (VarCode/VarIndex).
@param[in] ConnId   Connection identifier for the connection. 
                    The connection identifier can be determined with SMI_Login() or SMI_Connect().
@param[in] VarCode  Specifies which type of markers should be read.
                    - <tt>#Smi_MX_Code</tt>
                    - <tt>#Smi_MB_Code</tt>
                    - <tt>#Smi_MD_Code</tt>
                    - <tt>#Smi_MR_Code</tt>
                    - <tt>#Smi_MW_Code</tt>
                    - <tt>#Smi_RD_Code</tt>
                    - <tt>#Smi_GD_Code</tt>
@param[in] VarIndex Marker-Index
@retval #Smi_ERC_Ok OK
@retval #Smi_ERC_ConnId_InUse Other function is being processed.
@retval Smi_ERC_* Error codes are negative
*)
FUNCTION Smi_Read : DINT		(* Return: 0: OK, 1,2: BUSY, ErrorCode otherwise *)
VAR_INPUT
	ValAddr: DWORD;		(* Address to store read Value *)
	ConnId: DWORD;		(* Connection-Id *)
	VarCode: DWORD;		(* 1: MX, 2: MB, 3: MD, 4: MR, 5: MW *)
	VarIndex: DWORD;	(* Marker-Index *)
END_VAR
LD 0
END_FUNCTION

(* POU SMI_ReadBlock, ST *)
(**
@brief Reads a block of markers from a SMI-Module
@param[in] Req      Request enable
@param[in] ConnId   Connection identifier for the connection. 
                    The connection identifier can be determined with SMI_Login() or SMI_Connect().
@param[in] VarCode  Specifies which type of markers should be read.
                    - <tt>#Smi_MX_Code</tt>
                    - <tt>#Smi_MB_Code</tt>
                    - <tt>#Smi_MD_Code</tt>
                    - <tt>#Smi_MR_Code</tt>
                    - <tt>#Smi_MW_Code</tt>
                    - <tt>#Smi_RD_Code</tt>
                    - <tt>#Smi_GD_Code</tt>
@param[in] VarStart Marker-Index, determines the starting marker in the block.
@param[in] NumberOf Determines the size of the block, max. 256
@param[out] Ndr     TRUE if new data received
@param[out] Error   TRUE in case of error
@param[out] Status  Error code in case of error
                    - <tt>#Smi_ERC_Ok</tt> OK. <tt>Ndr = TRUE</tt>, result valid
                    - <tt>#Smi_ERC_Busy</tt> Completion/response is pending, result is not available
                    - <tt>Smi_ERC_*</tt> Error codes are negative. 
@param[out] Rdf     Data receive field
*)
FUNCTION_BLOCK SMI_ReadBlock
VAR_INPUT
	Req		: BOOL;
	ConnId	: DWORD;
	VarCode	: DWORD;
	VarStart	: DWORD;
	NumberOf : DINT;
END_VAR
VAR_OUTPUT
	Ndr		: BOOL;
	Error	 	: BOOL;
	Status		: DINT;
	Rdf 		: ARRAY[0..255] OF DWORD;
END_VAR
VAR
	fi: UDINT;
END_VAR
;
END_FUNCTION_BLOCK

(* POU SMI_ReadList, IL *)
(**
@brief Reads a list of markers from a SMI-Module
@param[in] Req Request enable
@param[in] ConnId Connection identifier for the connection. 
           The connection identifier can be determined with SMI_Login() or SMI_Connect().
@param[in] VAddrF Array with all markers which should be read.
@param[in] NumberOf Determines the number of markers (scope of list), maximal 64 
@param[out] Ndr TRUE if new data received
@param[out] Error TRUE in case of error
@param[out] Status Error code in case of error
    - <tt>#Smi_ERC_Ok</tt> OK. <tt>Ndr = TRUE</tt>, result valid
    - <tt>#Smi_ERC_Busy</tt> Completion/response is pending, result is not available
    - <tt>Smi_ERC_*</tt> Error codes are negative. 
@param[out] Rdf Data receive field
*)
FUNCTION_BLOCK SMI_ReadList
VAR_INPUT
	Req			: BOOL;
	ConnId		: DWORD;
	VAddrF	 	: ARRAY[0..63] OF VAR_ADDR;
	NumberOf 	: DINT;
END_VAR
VAR_OUTPUT
	Ndr			: BOOL;
	Error	 	: BOOL;
	Status	 	: DINT;
	Rdf 		: ARRAY[0..63] OF DWORD;
END_VAR
VAR
	fi: UDINT;
END_VAR
LD 0
END_FUNCTION_BLOCK

(* POU SMI_ReadString, ST *)
(**
@brief Reads a String or Stream of Bytes from a SMI-Module
@param[in]  Req    Request enable
@param[in]  ConnId Connection identifier for the connection. 
                   The connection identifier can be determined with SMI_Login() or SMI_Connect().
@param[in]  VAddr  Specifies which SVI Variable should be read.
                   VAR_ADDR can be determined with SMI_GetAddress().
@param[in]  Addr   Address of your buffer as the destination for the data.
                   Use the ADR() operator to get the address of your buffer.
@param[in]  Length Maximum number of bytes that can be written to the destination buffer.
                   Use the SIZEOF() operator to get the size of your buffer.
@param[out] Ndr    TRUE if new data received
@param[out] Error  TRUE in case of error
@param[out] Status Error code in case of error
                   - <tt>#Smi_ERC_Ok</tt> OK. <tt>Ndr = TRUE</tt>, result valid
                   - <tt>#Smi_ERC_Busy</tt> Completion/response is pending, result is not available
                   - <tt>Smi_ERC_*</tt> Error codes are negative 
@param[out] NRead  Number of bytes successfully read from the source and written to the destination buffer.
*)
FUNCTION_BLOCK SMI_ReadString
VAR_INPUT
	Req			: BOOL;
	ConnId		: DWORD;
	VAddr		: VAR_ADDR;
	Addr 		: DWORD;
	Length		: UINT;
END_VAR
VAR_OUTPUT
	Ndr			: BOOL;
	Error	 	: BOOL;
	Status		: DINT;
	NRead		: UINT;
END_VAR
VAR
	fi: UDINT;
END_VAR
;
END_FUNCTION_BLOCK

(* POU SMI_ReadVar, ST *)
(**
@brief Reads a SVI variable from a SMI-Module
@param[in] Req       Request enable
@param[in] ConnId    Connection identifier for the connection. 
                     The connection identifier can be determined with SMI_Login() or SMI_Connect().
@param[in]  VAddr    Specifies which SVI Variable should be read.
                     VAR_ADDR can be determined with SMI_GetAddress().
@param[out] Ndr      TRUE if new data received
@param[out] Error    TRUE in case of error
@param[out] Status   Error code in case of error
                     - <tt>#Smi_ERC_Ok</tt> OK. <tt>Ndr = TRUE</tt>, result valid
                     - <tt>#Smi_ERC_Busy</tt> Completion/response is pending, result is not available
                     - <tt>Smi_ERC_*</tt> Error codes are negative 
@param[out] IntegVal Read-value if Integer
@param[out] FloatVal Read-value if Floating-Point
*)
FUNCTION_BLOCK SMI_ReadVar
VAR_INPUT
	Req			: BOOL;
	ConnId		: DWORD;
	VAddr		: VAR_ADDR;
END_VAR
VAR_OUTPUT
	Ndr			: BOOL;
	Error	 	: BOOL;
	Status		: DINT;
	IntegVal	: DWORD;
	FloatVal	: REAL;
END_VAR
VAR
	fi: UDINT;
END_VAR
;
END_FUNCTION_BLOCK

(* POU SMI_ReleaseAccess, ST *)
(**
@brief The logged on user can release his active write authorization by means of this function.
       If access management with the keyword AccessHandler is configured in mconfig.ini under (SysMode), 
       the request to check and activate write authorization is passed on to access management.
@param[in] Req Request enable
@param[in] ConnId Transfer of the connection identifier for the connection. The identifier can be determined 
	with SMI_Login() or SMI_Connect().
@param[out] Done TRUE if ready
@param[out] Error TRUE in case of error
@param[out] Status Error code in case of error 
    - <tt>#Smi_ERC_Ok</tt> OK. <tt>Done = TRUE</tt>, Result valid
    - <tt>#Smi_ERC_Busy</tt> Completion/response is pending, Result is not available- <tt>Smi_ERC_*</tt> Error codes are negative.
*)
FUNCTION_BLOCK SMI_ReleaseAccess
VAR_INPUT
	Req: BOOL;
	ConnId: DWORD;
END_VAR
VAR_OUTPUT
	Done: BOOL;
	Error: BOOL;
	Status: DINT;
END_VAR
VAR
	fi: UDINT;
END_VAR
;
END_FUNCTION_BLOCK

(* POU SMI_RequestAccess, ST *)
(**
@brief The logged on user can request enabled SVI write authorization by means of this function.
       The keyword AccessControl is used for activation in mconfig.ini under (SysMode).
       If the user priority is higher than that of the active user, the authorization is withdrawn
       and assigned to the new user.
       If access management with the keyword AccessHandler is configured in mconfig.ini under (SysMode), 
       the request to check and activate write authorization is passed on to access management.
@param[in] Req Request enable
@param[in] ConnId Transfer of the connection identifier for the connection. The identifier can be determined 
	with SMI_Login() or SMI_Connect().
@param[out] Done TRUE if ready
@param[out] Error TRUE in case of error
@param[out] Status Error code in case of error 
    - <tt>#Smi_ERC_Ok</tt> OK. <tt>Done = TRUE</tt>, Result valid
    - <tt>#Smi_ERC_Busy</tt> Completion/response is pending, Result is not available- <tt>Smi_ERC_*</tt> Error codes are negative.
*)
FUNCTION_BLOCK SMI_RequestAccess
VAR_INPUT
	Req: BOOL;
	ConnId: DWORD;
END_VAR
VAR_OUTPUT
	Done: BOOL;
	Error: BOOL;
	Status: DINT;
END_VAR
VAR
	fi: UDINT;
END_VAR
;
END_FUNCTION_BLOCK

(* POU Smi_RetainExport, ST *)
(**
@brief Exports the retain memory of the current application to the given file.
Note: 
	- If the file already exists it will be overwritten.
    - The export of the retain data is only possible if the option Restore retain variables on change" under
      PLC Configuration/M1 Parameters is selected.

@param[in] Request Request flag to start the export.
@param[in] FileName File to which data are written. Nedds the full directory and 
	file name to export the data to.
@param[out] State indicates if zero that the request was finished and if
	not zero that the export finished with an error.
@param[out] Error Contains the number of the error if State is not 0 or 1.
	- #RETEXP_E_UNKNOWNERROR Undefined error.
	- #RETEXP_E_NOMEMORY Memory for data generation could not be allocated.
	- #RETEXP_E_MISSINGSTRUCTFILE File couldn't be read.
	- #RETEXP_E_RETAINDATACORRUPT Initialization of retain variables failed.
	- #RETEXP_E_FILECREATIONFAILED File could not be created/overwritten.
*)
FUNCTION_BLOCK Smi_RetainExport
VAR_INPUT
	Request:				BOOL;
	FileName:				STRING(83);
END_VAR
VAR_OUTPUT
	State:					DINT;
	Error:					BOOL;
END_VAR
VAR
	hJob: 					DWORD;
END_VAR
;
END_FUNCTION_BLOCK

(* POU SMI_SetBlk, ST *)
(**
@brief Writes a String or Stream of Bytes to SMI-Module
@param[in] Req Request enable
@param[in] ConnId Transfer of the connection identifier for the connection.
    The identifier to be transferred can be determined with SMI_Login() or SMI_Connect().
@param[in] SmiHandle Smi-Address-Handle, this is determined by SMI_GetAddr().
@param[in] Addr Contains the address of the values to be written.
@param[in] Length Indicates the length of the data block to be written (If a block of 
    markers is to be read, the value byte stream has to be 4-byte aligned).
@param[out] Done TRUE if operation successfully completed/data send
@param[out] Error TRUE in case of error
@param[out] Status see Smi_ERC_*
    - #Smi_ERC_Ok OK/Done
    - #Smi_ERC_Busy Completion/response is pending, result is not available
    - Smi_ERC_* Error occured
*)
FUNCTION_BLOCK SMI_SetBlk
VAR_INPUT
	Req			: BOOL;
	ConnId		: DWORD;
	SmiHandle	: SMI_ADDR;
	Addr 		: DWORD;
	Length		: UINT;
END_VAR
VAR_OUTPUT
	Done		: BOOL;
	Error		: BOOL;
	Status		: DINT;
END_VAR
VAR
	fi			: UDINT;
END_VAR
;
END_FUNCTION_BLOCK

(* POU SMI_SetVal, ST *)
(**
@brief Writes to a Marker/Variable of a SMI-Module
@param[in] Req Request enable
@param[in] ConnId Transfer of the connection identifier for the connection.
    The identifier to be transferred can be determined with SMI_Login() or SMI_Connect().
@param[in] SmiHandle 64-Bit Smi Object Handle/process value's address. This is determined 
	by SMI_GetAddr().
@param[in] Value Value to be written
@param[out] Done TRUE if operation successfully completed/data send
@param[out] Error TRUE in case of error
@param[out] Status see Smi_ERC_*
    - #Smi_ERC_Ok OK/Done
    - #Smi_ERC_Busy Completion/response is pending, result is not available
    - Smi_ERC_* Error occured
*)
FUNCTION_BLOCK SMI_SetVal
VAR_INPUT
	Req			: BOOL;
	ConnId		: DWORD;
	SmiHandle	: SMI_ADDR;
	Value		: DWORD;
END_VAR
VAR_OUTPUT
	Done		: BOOL;
	Error	 	: BOOL;
	Status		: DINT;
END_VAR
VAR
	fi			: UDINT;
END_VAR
;
END_FUNCTION_BLOCK

(* POU Smi_SetValFn, IL *)
(**
@brief Writes a Smi Object (specified by SmiAddr) of SMI-Module.
    Implementation: an Rpc-Request is done. Write may be BUSY
    until Rpc-Reply is received.
@param[in] ConnId Transfer of the connection identifier for the connection.
    The identifier to be transferred can be determined with SMI_Login() or SMI_Connect().
@param[in] SmiAddr Address of the 64-Bit Smi Object Handle/process value's address. 
	This is determined by SMI_GetAddr().
@param[in] ValAddr Address of the process value to be written
@retval #Smi_ERC_Ok OK
@retval #Smi_ERC_Busy Completion/response is pending; read value not available yet
@retval #Smi_ERC_ConnId_InUse Other function is being processed; communication in process
@retval Smi_ERC_* Error codes are negative 
*)
FUNCTION Smi_SetValFn : DINT
VAR_INPUT
	ConnId		: DWORD;
	SmiAddr		: DWORD;
	ValAddr		: DWORD;
END_VAR
	LD		0
END_FUNCTION

(* POU SMI_SetValLst, ST *)
(**
@brief Writes a List of Smi-Objects of SMI-Module
@param[in] Req Request enable
@param[in] ConnId Transfer of the connection identifier for the connection.
    The identifier to be transferred can be determined with SMI_Login() or SMI_Connect().
@param[in] SmiHandleF Array of process value addresses of the type SMI_ADDR.
    The process value addresses are determined with SMI_GetAddr().
@param[in] NumberOf Number of addresses, max. 64
@param[in] Sdf Data send field/values to be written
@param[out] Done TRUE if operation successfully completed/data send
@param[out] Error TRUE in case of error
@param[out] Status see Smi_ERC_*
    - #Smi_ERC_Ok OK/Done
    - #Smi_ERC_Busy Completion/response is pending, result is not available
    - Smi_ERC_* Error occured
*)
FUNCTION_BLOCK SMI_SetValLst
VAR_INPUT
	Req			: BOOL;
	ConnId		: DWORD;
	SmiHandleF  : ARRAY[0..63] OF SMI_ADDR;
	NumberOf 	: DINT;
	Sdf			: ARRAY[0..63] OF DWORD;
END_VAR
VAR_OUTPUT
	Done		: BOOL;
	Error	 	: BOOL;
	Status		: DINT;
END_VAR
VAR
	fi			: UDINT;
END_VAR
;
END_FUNCTION_BLOCK

(* POU Smi_SOCK_ClientOpen, ST *)
(**
@brief Opens a connection to a socket server. Address family of server
    must be AF_INET.
Note: The socket server must be running before this is called.
@param[in] ProtType Protocol of socket connection, see Smi_SOCK_Prot_*
@param[in] ServerPort Port of server, only needed at TCP
@param[in] ServerIP IP address of server, only needed at TCP
@param[in] Mode Mode of FB, see Smi_SOCK_Mode_*
@param[in] Req If false only state is returned. If true and state is not busy,
    a command is done.
@param[out] ConnDesc Connection description of socket communication
@param[out] State see Smi_ERC_Sock*
    - 0 OK/Done
    - Smi_ERC_Sock* Error occured
*)
FUNCTION_BLOCK Smi_SOCK_ClientOpen
VAR_INPUT
	ProtType:		DWORD;
	ServerPort:		WORD;
	ServerIP:		DINT;
	Mode:			DINT;
	Req:			BOOL;
END_VAR
VAR_OUTPUT
	State:			DINT;
	ConnDesc:		SMI_SOCK_CONTROL;
END_VAR
VAR
END_VAR
;
END_FUNCTION_BLOCK

(* POU Smi_SOCK_ClientOpen_NB, ST *)
(**
@brief Opens a connection to a socket server. Address family of server
    must be AF_INET.
  Note: The socket server must be running before this is called.
@param[in] ProtType Protocol of socket connection, see Smi_SOCK_Prot...
@param[in] ServerPort Port of server, only needed at TCP
@param[in] ServerIP IP address of server, only needed at TCP
@param[in] ClientIP IP address of client (which interface to use), can be empty.
@param[in] Req If false only state is returned. If true and state is not busy,
   a command is done.
@param[out] ConnDesc Connection Description of socket communication
@param[out] Done TRUE if operation successfully completed
@param[out] Error TRUE in case of error
@param[out] State see Smi_ERC_Sock*
    - Smi_ERC_Ok OK/Done
    - Smi_ERC_Busy Completion/response is pending, result is not available
    - Smi_ERC_Sock* Error occured
*)
FUNCTION_BLOCK Smi_SOCK_ClientOpen_NB
VAR_INPUT
	ProtType:		DWORD;
	ServerPort:		WORD;
	ServerIP:		DINT;
	ClientIP:       DINT;
	Req:			BOOL;
END_VAR
VAR_OUTPUT
	Done : BOOL;				(* TRUE => operation completed *)
	Error : BOOL;				(* TRUE in case of error *)
	State : DINT;				(* 0: OK/Done, 1: BUSY, Error-Code in case of error *)
	ConnDesc:		SMI_SOCK_CONTROL;
END_VAR
VAR
	Pltd : DWORD;
END_VAR
;
END_FUNCTION_BLOCK

(* POU Smi_SOCK_Close, ST *)
(**
@brief Closes a connection to a socket server or client. Only data member
    ProtType and Socket are used from input variable ConnDesc.
@param[in] ConnDesc Description of socket to close.
@param[in] Req If false only state is returned. If true and state is not busy,
    a command is done.
@param[out] State see Smi_ERC_Sock*
    - Smi_ERC_Ok OK/Done
    - Smi_ERC_Sock* Error occured
*)
FUNCTION_BLOCK Smi_SOCK_Close
VAR_INPUT
	ConnDesc:		SMI_SOCK_CONTROL;
	Req:			BOOL;
END_VAR
VAR_OUTPUT
	State:			DINT;
END_VAR
VAR
END_VAR
;
END_FUNCTION_BLOCK

(* POU Smi_SOCK_Close_NB, ST *)
(**
@brief Closes a connection to a socket server or client in non blocking mode. 
    Only data member ProtType and Socket are used from input variable ConnDesc.
@param[in] ConnDesc Description of socket to close.
@param[in] Req If false only state is returned. If true and state is not busy,
    a command is done.
@param[out] Done TRUE if operation successfully completed
@param[out] Error TRUE in case of error
@param[out] State see Smi_ERC_Sock*
    - Smi_ERC_Ok OK/Done
    - Smi_ERC_Busy Completion/response is pending, result is not available
    - Smi_ERC_Sock* Error occured
*)
FUNCTION_BLOCK Smi_SOCK_Close_NB
VAR_INPUT
	ConnDesc:		SMI_SOCK_CONTROL;
	Req:			BOOL;
END_VAR
VAR_OUTPUT
	Done: BOOL;
	Error: BOOL;
	State: DINT;
END_VAR
VAR
	PThread: DWORD;
END_VAR
;
END_FUNCTION_BLOCK

(* POU Smi_SOCK_Read, ST *)
(**
@brief Reads data from a socket connection.
    Note: This function is blocks the PLC cycle till data are received!
@param[in] ConnDesc socket of communication
@param[in] DataBuf Address of data buffer, use ADR()
@param[in] DataLen Length of data buffer
@param[in] Mode Mode of FB, see Smi_SOCK_Mode*
@param[in] Req If false only state is returned. If true and state is not busy,
    a command is done.
@param[out] RecLen Length of received data
@param[out] State see Smi_ERC_Sock*
    - Smi_ERC_Ok OK/Done
    - Smi_ERC_Sock* Error occured
@param[out] RecConnDesc Description of socket client, needed at a UDP server
*)
FUNCTION_BLOCK Smi_SOCK_Read
VAR_INPUT
	ConnDesc:		SMI_SOCK_CONTROL;
	Mode:			DINT;
	DataBuf:		DWORD;
	DataLen:		DINT;
	Req:			BOOL;
END_VAR
VAR_OUTPUT
	RecLen:			DINT;
	State:			DINT;
	RecConnDesc:	SMI_SOCK_CONTROL;
END_VAR
VAR
END_VAR
;
END_FUNCTION_BLOCK

(* POU Smi_SOCK_Read_NB, ST *)
(**
@brief Reads data from a socket connection in a non-blocking mode. 
@param[in] ConnDesc socket of communication
@param[in] DataBuf Address of data buffer, use ADR()
@param[in] DataLen Length of data buffer
@param[in] Req If false only state is returned. If true and state is not busy,
    a command is done.
@param[out] Done TRUE if operation successfully completed
@param[out] Error TRUE in case of error
@param[out] State see Smi_ERC_Sock*
    - Smi_ERC_Ok OK/Done
    - Smi_ERC_Busy Completion/response is pending, result is not available
    - Smi_ERC_Sock* Error occured
@param[out] RecLen Length of received data
@param[out] RecConnDesc Description of socket client, needed at a UDP server
*)
FUNCTION_BLOCK Smi_SOCK_Read_NB
VAR_INPUT
	ConnDesc: SMI_SOCK_CONTROL;
	DataBuf: DWORD;
	DataLen: DINT;
	Req: BOOL;
END_VAR
VAR_OUTPUT
	Done: BOOL;
	Error: BOOL;
	State: DINT;
	RecLen: DINT;
	RecConnDesc: SMI_SOCK_CONTROL;
END_VAR
VAR
	PThread: DWORD;
END_VAR
;
END_FUNCTION_BLOCK

(* POU Smi_SOCK_ServerOpen, ST *)
(**
@brief Opens a connection to a socket client. Address family of server must 
    be AF_INET. Note: At TCP this function blocks the PLC cycle till a TCP client is opened!
@param[in] ProtType Protocoll of socket connection, see Smi_SOCK_Prot...
@param[in] ServerPort port of server
@param[in] ServerIP IP address of server
@param[in] Mode Mode of FB, see Smi_SOCK_Mode...
@param[in] Req If false only state is returned. If true and state is not busy,
    a command is done.
@param[out] ServerSocket Socket ID of server. Use it to close a socket server.
@param[out] State see Smi_ERC_Sock*
    - Smi_ERC_Ok OK/Done
    - Smi_ERC_Sock* Error occured
@param[out] ConnDesc Connection description of the client. Only at TCP it is filled
    correct.
*)
FUNCTION_BLOCK Smi_SOCK_ServerOpen
VAR_INPUT
	ProtType:		DWORD;
	ServerPort:		WORD;
	ServerIP:		DINT;
	Mode:			DINT;
	Req:			BOOL;
END_VAR
VAR_OUTPUT
	State:			DINT;
	ServerSocket:	DINT;
	ConnDesc:		SMI_SOCK_CONTROL;
END_VAR
VAR
END_VAR
;
END_FUNCTION_BLOCK

(* POU Smi_SOCK_ServerOpen_NB, ST *)
(**
@brief Non-blocking version of SMI_SOCK_ServerOpen, opens a connection
    to a socket client. The read/write transfers to this client are
    non-blocking. Address family of server must be AF_INET.
@param[in] Req Request enable
@param[in] ProtType protocol of socket connection, see Smi_SOCK_Prot...
@param[in] ServerPort port of server
@param[in] ServerIP IP address of server (which interface to use), can be empty.
@param[out] Done TRUE if operation successfully completed
@param[out] Error TRUE in case of error
@param[out] State see Smi_ERC_Sock*
    - Smi_ERC_Ok OK/Done
    - Smi_ERC_Busy Completion/response is pending, result is not available
    - Smi_ERC_Sock* Error occured
@param[out] ServerSocket Socket ID of server. Use it to close a socket server.
@param[out] ConnDesc Connection description of the client. Only at TCP it is filled
    correct.
*)
FUNCTION_BLOCK Smi_SOCK_ServerOpen_NB
VAR_INPUT
	ProtType:		DWORD;
	ServerPort:		WORD;
	ServerIP:		DINT;
	Req:			BOOL;
END_VAR
VAR_OUTPUT
	Done : BOOL;				(* TRUE => operation completed *)
	Error : BOOL;				(* TRUE in case of error *)
	State : DINT;				(* 0: OK/Done, 1: BUSY, Error-Code in case of error *)
	ServerSocket:	DINT;
	ConnDesc:		SMI_SOCK_CONTROL;
END_VAR
VAR
	Pltd : DWORD;
END_VAR
;
END_FUNCTION_BLOCK

(* POU Smi_SOCK_SetOpt, ST *)
(**
@brief This function block sets the options associated with a socket
    connection. Only 'socket level' options (SOL_SOCKET) are
    performed (see also setsockopt() VxWorks).
    Note: The socket server must be running before this is called.
@param[in] ConnDesc Connection Description of socket communication
@param[in] OptName Name of option to be set, see Smi_SOCK_SO_*
@param[in] OptVal New value of option to be set
@param[in] Req If false only state is returned. If true and state is not busy,
    a command is done.
@param[out] State see Smi_ERC_Sock*
    - Smi_ERC_Ok OK/Done
    - Smi_ERC_Sock* Error occured
*)
FUNCTION_BLOCK Smi_SOCK_SetOpt
VAR_INPUT
	ConnDesc:		SMI_SOCK_CONTROL;
	OptName:		DINT;
	OptVal:			DINT;
	Req:			BOOL;
END_VAR
VAR_OUTPUT
	State:			DINT;

END_VAR
VAR
END_VAR
;
END_FUNCTION_BLOCK

(* POU Smi_SOCK_Write, ST *)
(**
@brief Writes to a socket connection.
@param[in] ConnDesc Description of the socket partner
@param[in] DataBuf Address of data buffer, use ADR()
@param[in] DataLen Length of data buffer
@param[in] Mode Mode of FB, see Smi_SOCK_Mode...
@param[in] Req If false only state is returned. If true and state is not busy,
    a command is done.
@param[out] SendLen Lenght of sended data
@param[out] State see Smi_ERC_Sock*
    - Smi_ERC_Ok OK/Done
    - Smi_ERC_Busy Completion/response is pending, result is not available
    - Smi_ERC_Sock* Error occured
*)
FUNCTION_BLOCK Smi_SOCK_Write
VAR_INPUT
	ConnDesc:		SMI_SOCK_CONTROL;
	DataBuf:		DWORD;
	DataLen:		DINT;
	Mode:			DINT;
	Req:			BOOL;
END_VAR
VAR_OUTPUT
	State:			DINT;
	SendLen:		DINT;
END_VAR
VAR
END_VAR
;
END_FUNCTION_BLOCK

(* POU Smi_SOCK_Write_NB, ST *)
(**
@brief Writes to a socket connection in a non-blocking mode. 
@param[in] ConnDesc Description of the socket partner
@param[in] DataBuf Address of data buffer, use ADR()
@param[in] DataLen Length of data buffer
@param[in] Mode Mode of FB, see Smi_SOCK_Mode...
@param[in] Req If false only state is returned. If true and state is not busy,
    a command is done.
@param[out] Done TRUE if operation successfully completed
@param[out] Error TRUE in case of error
@param[out] State see Smi_ERC_Sock*
    - Smi_ERC_Ok OK/Done
    - Smi_ERC_Busy Completion/response is pending, result is not available
    - Smi_ERC_Sock* Error occured
@param[out] SendLen Lenght of sended data
*)
FUNCTION_BLOCK Smi_SOCK_Write_NB
VAR_INPUT
	ConnDesc: SMI_SOCK_CONTROL;
	DataBuf: DWORD;
	DataLen: DINT;
	Req: BOOL;
END_VAR
VAR_OUTPUT
	Done: BOOL;
	Error: BOOL;
	State: DINT;
	SendLen: DINT;
END_VAR
VAR
	PThread: DWORD;
END_VAR
;
END_FUNCTION_BLOCK

(* POU Smi_SOCK_WriteTo, ST *)
(**
@brief Writes to a socket connection.
@param[in] ConnDesc Description of the socket partner
@param[in] ServerPort Port of server
@param[in] ServerIP IP address of server
@param[in] DataBuf Address of data buffer, use ADR()
@param[in] DataLen Length of data buffer
@param[in] Mode Mode of FB, see Smi_SOCK_Mode...
@param[in] Req If false only state is returned. If true and state is not busy,
    a command is done.
@param[out] SendLen Lenght of sended data
@param[out] State see Smi_ERC_Sock*
    - Smi_ERC_Ok OK/Done
    - Smi_ERC_Busy Completion/response is pending, result is not available
    - Smi_ERC_Sock* Error occured
*)
FUNCTION_BLOCK Smi_SOCK_WriteTo
VAR_INPUT
	ConnDesc:		SMI_SOCK_CONTROL;
	ServerPort:		WORD;
	ServerIP:		DINT;
	DataBuf:		DWORD;
	DataLen:		DINT;
	Mode:			DINT;
	Req:			BOOL;
END_VAR
VAR_OUTPUT
	State:			DINT;
	SendLen:		DINT;
END_VAR
VAR
END_VAR
;
END_FUNCTION_BLOCK

(* POU Smi_SOCK_WriteTo_NB, ST *)
(**
@brief Writes to a socket connection in a non blocking mode. 
@param[in] ConnDesc Description of the socket partner
@param[in] ServerPort Port of server
@param[in] ServerIP IP address of server
@param[in] DataBuf Address of data buffer, use ADR()
@param[in] DataLen Length of data buffer
@param[in] Req If false only state is returned. If true and state is not busy,
    a command is done.
@param[out] Done TRUE if operation successfully completed
@param[out] Error TRUE in case of error
@param[out] State see Smi_ERC_Sock*
    - Smi_ERC_Ok OK/Done
    - Smi_ERC_Busy Completion/response is pending, result is not available
    - Smi_ERC_Sock* Error occured
@param[out] SendLen Lenght of sended data
*)
FUNCTION_BLOCK Smi_SOCK_WriteTo_NB
VAR_INPUT
	ConnDesc: SMI_SOCK_CONTROL;
	ServerPort: WORD;
	ServerIP: DINT;
	DataBuf: DWORD;
	DataLen: DINT;
	Req: BOOL;
END_VAR
VAR_OUTPUT
	Done: BOOL;
	Error: BOOL;
	State: DINT;
	SendLen: DINT;
END_VAR
VAR
	PThread: DWORD;
END_VAR
;
END_FUNCTION_BLOCK

(* POU Smi_Write, IL *)
(**
@brief Writes Marker (specified by VarCode/VarIndex) of a SMI-Module
@param[in] ValAddr  Address of Value to write. Using the ADR operator, ValAddr 
                    must be created from the variable that contains the value to be written. 
                    This variable must comply with the specified market type (VarCode).
@param[in] ConnId   Connection identifier for the connection. 
                    The connection identifier can be determined with SMI_Login() or SMI_Connect().
@param[in] VarCode  Specifies which type of markers should be read.
                    - <tt>#Smi_MX_Code</tt>
                    - <tt>#Smi_MB_Code</tt>
                    - <tt>#Smi_MD_Code</tt>
                    - <tt>#Smi_MR_Code</tt>
                    - <tt>#Smi_MW_Code</tt>
                    - <tt>#Smi_RD_Code</tt>
                    - <tt>#Smi_GD_Code</tt>
@param[in] VarIndex Determines the marker index.
@retval #Smi_ERC_Ok OK
@retval #Smi_ERC_ConnId_InUse Other function is being processed
@retval Smi_ERC_* Error codes are negative
*)
FUNCTION Smi_Write : DINT
VAR_INPUT
	ValAddr:	DWORD;
	ConnId:		DWORD;
	VarCode: 	DWORD;
	VarIndex: 	DWORD;
END_VAR
	LD		0
END_FUNCTION

(* POU SMI_WriteBlock, ST *)
(**
@brief Writes to a Block of Markers of a SMI-Module
@param[in]  Req      Request enable
@param[in]  ConnId   Connection identifier for the connection. 
                     The connection identifier can be determined with SMI_Login() or SMI_Connect().
@param[in]  VarCode  Specifies which type of markers should be read.
                     - <tt>#Smi_MX_Code</tt>
	                 - <tt>#Smi_MB_Code</tt>
	                 - <tt>#Smi_MD_Code</tt>
	                 - <tt>#Smi_MR_Code</tt>
	                 - <tt>#Smi_MW_Code</tt>
	                 - <tt>#Smi_RD_Code</tt>
	                 - <tt>#Smi_GD_Code</tt>
@param[in]  VarStart Determines the starting marker in the block. 
@param[in]  NumberOf Determines the number of markers (size of Block), max. 256
@param[in]  Sdf      Data send field/values to be written.
@param[out] Done     TRUE if operation successfully completed
@param[out] Error    TRUE in case of error
@param[out] Status   Error code in case of error
                     - <tt>#Smi_ERC_Ok</tt> OK. <tt>Ndr = TRUE</tt>, result valid
                     - <tt>#Smi_ERC_Busy</tt> Completion/response is pending, result is not available
                     - <tt>Smi_ERC_*</tt> Error codes are negative 
*)
FUNCTION_BLOCK SMI_WriteBlock
VAR_INPUT
	Req			: BOOL;
	ConnId		: DWORD;
	VarCode		: DWORD;
	VarStart	: DWORD;
	NumberOf	: DINT;
	Sdf		 	: ARRAY[0..255] OF DWORD;
END_VAR
VAR_OUTPUT
	Done		: BOOL;
	Error	 	: BOOL;
	Status	 	: DINT;	
END_VAR
VAR
	fi: UDINT;
END_VAR
;
END_FUNCTION_BLOCK

(* POU SMI_WriteList, ST *)
(**
@brief Writes a List of Markers of a SMI-Module
@param[in]  Req      Request enable
@param[in]  ConnId   Connection identifier for the connection. 
                     The connection identifier can be determined with SMI_Login() or SMI_Connect().
@param[in]  VAddrF   Array with all markers which should be written.
@param[in]  NumberOf Number of Markers, max. 64
@param[in]  Sdf      Data send field/values to be written
@param[out] Done     TRUE if operation successfully completed
@param[out] Error    TRUE in case of error
@param[out] Status   Error code in case of error
                     - <tt>#Smi_ERC_Ok</tt> OK. <tt>Ndr = TRUE</tt>, result valid
                     - <tt>#Smi_ERC_Busy</tt> Completion/response is pending, result is not available
                     - <tt>Smi_ERC_*</tt> Error codes are negative 
*)
FUNCTION_BLOCK SMI_WriteList
VAR_INPUT
	Req			: BOOL;
	ConnId		: DWORD;
	VAddrF	 	: ARRAY[0..63] OF VAR_ADDR;
	NumberOf 	: DINT;
	Sdf			: ARRAY[0..63] OF DWORD;
END_VAR
VAR_OUTPUT
	Done		: BOOL;
	Error	 	: BOOL;
	Status		: DINT;
END_VAR
VAR
	fi			: UDINT;
END_VAR
;
END_FUNCTION_BLOCK

(* POU SMI_WriteString, ST *)
(**
@brief Writes a string or stream of bytes to a SMI-Module
@param[in]  Req    Request enable
@param[in]  ConnId Connection identifier for the connection. 
                   The connection identifier can be determined with SMI_Login() or SMI_Connect().
@param[in]  VAddr  Specifies which SVI Variable should be written.
                   VAR_ADDR can be determined with SMI_GetAddress().
@param[in]  Addr   Address of your buffer which contains the data to be written.
                   Use the ADR() operator to get the address of your buffer.
@param[in]  Length Number of bytes that should be written. For a STRING, the number 
                   of bytes can be calculated with LEN()+1 or the value 0 is used, whereby the calculation 
                   is executed by the function block itself. 
@param[out] Done   TRUE if operation successfully completed
@param[out] Error  TRUE in case of error
@param[out] Status Error code in case of error
                   - <tt>#Smi_ERC_Ok</tt> OK. <tt>Ndr = TRUE</tt>, result valid
                   - <tt>#Smi_ERC_Busy</tt> Completion/response is pending, result is not available
                   - <tt>Smi_ERC_*</tt> Error codes are negative 
*)
FUNCTION_BLOCK SMI_WriteString
VAR_INPUT
	Req			: BOOL;
	ConnId		: DWORD;
	VAddr		: VAR_ADDR;
	Addr 		: DWORD;
	Length		: UINT;
END_VAR
VAR_OUTPUT
	Done		: BOOL;
	Error		: BOOL;
	Status		: DINT;
END_VAR
VAR
	fi			: UDINT;
END_VAR
;
END_FUNCTION_BLOCK

(* POU SMI_WriteVar, ST *)
(**
@brief Writes a SVI variable of a SMI-Module
@param[in]  Req      Request enable
@param[in]  ConnId   Connection identifier for the connection. 
                     The connection identifier can be determined with SMI_Login() or SMI_Connect().
@param[in]  VAddr    Specifies which SVI Variable should be written.
                     VAR_ADDR can be determined with SMI_GetAddress().
@param[in]  IntegVal Write-value: if an integer, bit or byte value is expected, 
                     this must be specified here
@param[in]  FloatVal Write-Value: if a foating point value is expected, this 
                     must be specified here.
@param[out] Done     TRUE if operation successfully completed
@param[out] Error    TRUE in case of error
@param[out] Status   Error code in case of error
                     - <tt>#Smi_ERC_Ok</tt> OK. <tt>Ndr = TRUE</tt>, result valid
                     - <tt>#Smi_ERC_Busy</tt> Completion/response is pending, result is not available
                     - <tt>Smi_ERC_*</tt> Error codes are negative 
*)
FUNCTION_BLOCK SMI_WriteVar
VAR_INPUT
	Req			: BOOL;
	ConnId		: DWORD;
	VAddr		: VAR_ADDR;
	IntegVal	: DWORD;
	FloatVal	: REAL;
END_VAR
VAR_OUTPUT
	Done		: BOOL;
	Error	 	: BOOL;
	Status		: DINT;
END_VAR
VAR
	fi			: UDINT;
END_VAR
;
END_FUNCTION_BLOCK
